FUNCTION_BLOCK fb_add
VAR_INPUT
	in1:INT;
	in2:INT;
END_VAR
VAR_OUTPUT
	out:INT;
	
END_VAR
VAR
END_VAR


out :=in1+in2;

END_FUNCTION_BLOCK

(* stored: Version 1.1.0.1, ProductVersion 3.1.4024.9
   POU fb_add: Id {8681f88c-fa23-4638-9887-de06f9eedc1d}, SpecialFunc None *)
